(* Logix 5000 project; controller WWTP_SOLIDS_CLX vendor 1 type 14 code 54 rev 17.2; software revision 17.00; part 5 of 16 *)
(* tags used below, declared in another part *)
   Inp_RatePVBad : BOOL;   // 1=Rate PV Input Quality = Bad (fail)
   Inp_RatePVUncertain : BOOL;   // 1=Rate PV Input Quality = Uncertain
   Inp_QtyPVBad : BOOL;   // 1=Quantity PV Input Quality = Bad (fail)
   Inp_QtyPVUncertain : BOOL;   // 1=Quantity PV Input Quality = Uncertain
   Inp_CtrldEqpFault : BOOL;   // Controlled Equipment device or I/O status 0=OK, 1=fail
   Inp_Sim : BOOL;   // 1=Simulate working flowmeter; 0=use actual flowmeter
   Cfg_HasDribble : BOOL;   // 1=Slow to Dribble before complete, 0=use complete only
   Cfg_CalcRate : BOOL;   // 1=differentiate Inp_Qty to get rate, 0=use Inp_Rate
   Cfg_CalcQty : BOOL;   // 1=integrate Inp_Rate to get Quantity, 0=use Inp_Qty
   Cfg_PCmdClear : BOOL;   // 1=Clear Program Commands on receipt 0=Leave Set
   Cfg_HasOverTolAlm : BOOL;   // 1=Over Tolerance Alarm exists and will be checked
   Cfg_HasUnderTolAlm : BOOL;   // 1=Under Tolerance Alarm exists and will be checked
   Cfg_HasZeroFaultAlm : BOOL;   // 1=Zero Fault Alarm exists and will be checked
   Cfg_HasEqpFaultAlm : BOOL;   // 1=Equipment Fault Alarm exists and will be checked
   Cfg_OverTolResetReqd : BOOL;   // 1=Reset requied to clear Out of Tolerance High Alarm
   Cfg_UnderTolResetReqd : BOOL;   // 1=Reset required to clear Out of Tolerance Low Alarm
   Cfg_ZeroFaultResetReqd : BOOL;   // 1=Reset required to clear Zero Fault Alarm
   Cfg_EqpFaultResetReqd : BOOL;   // 1=Reset required to clear Equipment Fault Alarm
   Cfg_OverTolAckReqd : BOOL;   // 1=Acknowledge required for Out of Tolerance High Alarm
   Cfg_UnderTolAckReqd : BOOL;   // 1=Acknowledge required for Out of Tolerance Low Alarm
   Cfg_ZeroFaultAckReqd : BOOL;   // 1=Acknowledge required for Zero Fault Alarm
   Cfg_EqpFaultAckReqd : BOOL;   // 1=Acknowledge required for Equipment Fault Alarm
   Cfg_OverTolSeverity : SINT;   // Over Tolerance Alarm Severity 1=info, 2=warn, 3=excep, 4=fault
   Cfg_UnderTolSeverity : SINT;   // Under Tolerance Alarm Severity 1=info, 2=warn, 3=excep, 4=fault
   Cfg_ZeroFaultSeverity : SINT;   // Zero Fault Alarm Severity 1=info, 2=warn, 3=excep, 4=fault
   Cfg_EqpFaultSeverity : SINT;   // Equipment Fault Alarm Severity 1=info, 2=warn, 3=excep, 4=fault
   Cfg_MaxQty : REAL;   // Maximum allowed quantity to deliver (setpoint) (EU)
   Cfg_EUQtyMult : REAL;   // Rate to Quantity EU Multiplier (e.g., Gal to Bbl.)
   Cfg_Rollover : REAL;   // Quantity Rollover (e.g., total counts for pulse input)
   Cfg_CountsPerEU : REAL;   // Number of Counts in Inp_QtyPV which equal 1.0 EU
   Cfg_RateTime : REAL;   // Time factor for rate (60 for /min, 3600 for /hr) (Sec)
   Cfg_RateFiltTC : REAL;   // Filter Time Constant (sec) for calculated Rate
   Cfg_LoRateCutoff : REAL;   // Rate below which to report zero flow (Inp_RatePV untis)
   Cfg_SimRate : REAL;   // Rate at which to deliver when running in Simulation (EU/rate time)
   Cfg_SimDribbleRate : REAL;   // Rate at which to dribble when running in Simulation (EU/rate time)
   PCmd_OverTolAck : BOOL;   // Program Command to Acknowledge Out of Tolerance High Alarm
   PCmd_OverTolInhibit : BOOL;   // Program Command to Inhibit Out of Tolerance High Alarm
   PCmd_OverTolUninhibit : BOOL;   // Program Command to Uninhibit Out of Tolerance High Alarm
   PCmd_UnderTolAck : BOOL;   // Program Command to Acknowledge Out of Tolerance Low Alarm
   PCmd_UnderTolInhibit : BOOL;   // Program Command to Inhibit Out of Tolerance Low Alarm
   PCmd_UnderTolUninhibit : BOOL;   // Program Command to Uninhibit Out of Tolerance Low Alarm
   PCmd_ZeroFaultAck : BOOL;   // Program Command to Acknowledge Zero Fault Alarm
   PCmd_ZeroFaultInhibit : BOOL;   // Program Command to Inhibit Zero Fault Alarm
   PCmd_ZeroFaultUninhibit : BOOL;   // Program Command to Uninhibit Zero Fault Alarm
   PCmd_EqpFaultAck : BOOL;   // Program Command to Acknowledge Equipment Fault Alarm
   PCmd_EqpFaultInhibit : BOOL;   // Program Command to Inhibit Equipment Fault Alarm
   PCmd_EqpFaultUninhibit : BOOL;   // Program Command to Uninhibit Equipment Fault Alarm
   Out_RunFlow : BOOL;   // 1=Deliver at Full (fast) Flow
   Out_DribbleFlow : BOOL;   // 1=Deliver at Dribble (slow) Flow
   Out_StopFlow : BOOL;   // 1=Stop Delivery Equipment
   Out_RunTot : BOOL;   // 1=Run external totalizer (e.g. onboard flowmeter)
   Val_Qty : REAL;   // Quantity actually delivered (totalizer output) (EU)
   Val_SP : REAL;   // Amount to be delivered (Setpoint) (EU)
   Val_DribbleQty : REAL;   // Amount to be delivered at slow rate (EU)
   Val_Preact : REAL;   // Amount before SP at which flow will be stopped (EU)
   Val_Notify : SINT;   // Current Alarm Level and Acknowledgement (enumeration)
   Sts_Cleared : BOOL;   // 1=Totalizer Clear completed
   Sts_TotRunning : BOOL;   // 1=Totalizer Running, 0=Totalizer Stopped
   Sts_FlowRunning : BOOL;   // 1=Flow is Running (Out_Run is ON)
   Sts_FlowDribble : BOOL;   // 1=Flow is slowed to Dribble (Out_Dribble is ON)
   Sts_FlowStopped : BOOL;   // 1=Flow is Stopped (Out_Stop is ON)
   Sts_Bumping : BOOL;   // 1=Bump flow (timed) is active
   Sts_Complete : BOOL;   // 1=Total Delivered > (SP - Preact)
   Sts_Available : BOOL;   // 1=Dosing available for control by automation (Prog)
   Sts_QtyBad : BOOL;   // 1=Quantity Value is Bad (PV Fail)
   Sts_QtyUncertain : BOOL;   // 1=Quantity Value is Uncertain
   Sts_RateBad : BOOL;   // 1=Rate Value is Bad (PV Fail)
   Sts_RateUncertain : BOOL;   // 1=Rate Value is Uncertain
   Sts_Err : BOOL;   // 1=Error: Bad Configuration, see detail Err bits for reason
   Err_EU : BOOL;   // 1=Error: Cfg_CountsPerEU, Cfg_EUQtyMult or Cfg_Rollowver invalid
   Err_Rate : BOOL;   // 1=Error: Cfg_RateFiltTC or Cfg_RateTime invalid
   Err_Cutoff : BOOL;   // 1=Error: Cfg_LoRateCutoff invalid
   Err_Limit : BOOL;   // 1=Error: Cfg_MaxQty invalid
   Err_Sim : BOOL;   // 1=Error: Cfg_SimDribbleRate or Cfg_SimRate invalid
   Err_Timer : BOOL;   // 1=Error: Cfg_BumpT or Cfg_ClearPulseT (use 0.0 to 2147483.647)
   Err_Alarm : BOOL;   // 1=Error: Alarm Severity Cfg Invalid
   Sts_Maint : BOOL;   // 1=Mode is Maintenance (supersedes Prog, Oper)
   Sts_Prog : BOOL;   // 1=Mode is Program (auto)
   Sts_Oper : BOOL;   // 1=Mode is Operator (manual)
   Sts_ProgOperLock : BOOL;   // 1=Program or Operator has requested Mode Lock
   Sts_OverTol : BOOL;   // 1=Delivery Out of Tolerance High
   Alm_OverTol : BOOL;   // 1=Delivery Out of Tolerance High Alarm
   Ack_OverTol : BOOL;   // 1=Out of Tolerance High Alarm has been acknowledged
   Sts_OverTolDisabled : BOOL;   // 1=Out of Tolerance High Alarm has been disabled (will not be sent)
   Sts_OverTolInhibited : BOOL;   // 1=Out of Tolerance High Alarm has been inhibited by logic
   Sts_OverTolSuppressed : BOOL;   // 1=Out of Tolerance High Alarm has been suppressed (logged only)
   Sts_UnderTol : BOOL;   // 1=Delivery Out of Tolerance Low
   Alm_UnderTol : BOOL;   // 1=Delivery Out of Tolerance Low Alarm
   Ack_UnderTol : BOOL;   // 1=Out of Tolerance Low Alarm has been acknowledged
   Sts_UnderTolDisabled : BOOL;   // 1=Out of Tolerance Low Alarm has been disabled (will not be sent)
   Sts_UnderTolInhibited : BOOL;   // 1=Out of Tolerance Low Alarm has been inhibited by logic
   Sts_UnderTolSuppressed : BOOL;   // 1=Out of Tolerance Low Alarm has been suppressed (logged only)
   Sts_ZeroFault : BOOL;   // 1=Total did not clear or unexpected flow
   Alm_ZeroFault : BOOL;   // 1=Warning: Total did not clear or still flowing
   Ack_ZeroFault : BOOL;   // 1=Zero Fault Alarm has been acknowledged
   Sts_ZeroFaultDisabled : BOOL;   // 1=Zero Fault Alarm is Disabled (not saved or sent)
   Sts_ZeroFaultInhibited : BOOL;   // 1=Zero Fault Alarm has been inhibited by logic
   Sts_ZeroFaultSuppressed : BOOL;   // 1=Zero Fault Alarm has been suppressed (logged only)
   Sts_EqpFault : BOOL;   // 1=Equipment Fault Detected
   Alm_EqpFault : BOOL;   // 1=Equipment Fault Alarm
   Ack_EqpFault : BOOL;   // 1=Equipment Fault Alarm has been acknowledged
   Sts_EqpFaultDisabled : BOOL;   // 1=Equipment Fault Alarm is Disabled (not saved or sent)
   Sts_EqpFaultInhibited : BOOL;   // 1=Equipment Fault Alarm has been inhibited by logic
   Sts_EqpFaultSuppressed : BOOL;   // 1=Equipment Fault Alarm has been suppressed (logged only)
   Rdy_ClearTot : BOOL;   // 1=Ready for OCmd_ClearTot (enables button)
   Rdy_StartTot : BOOL;   // 1=Ready for OCmd_StartTot (enables button)
   Rdy_StopTot : BOOL;   // 1=Ready for OCmd_StopTot (enables button)
   Rdy_StartFlow : BOOL;   // 1=Ready for OCmd_StartFlow (enables button)
   Rdy_StopFlow : BOOL;   // 1=Ready for OCmd_StopFlow (enables button)
   Rdy_CheckTol : BOOL;   // 1-Ready for OCmd_CheckTol (enables button)
   Rdy_Bump : BOOL;   // 1=Ready for OCmd_Bump (enables button)
   Rdy_Reset : BOOL;   // 1=Ready for OCmd_Reset (enables button)
   Wrk_Notify : DINT;   // Buffer for building Val_Notify
   Mode : P_Mode;   // Analog Input Mode Selection
   Wrk_ClearTot : BOOL;   // Request to Clear Total received
   ZeroFault : P_Alarm;   // Rate Not Zero when Expected Alarm
   UnderTol : P_Alarm;   // Final Quantity Below Low Tolerance Alarm
   OverTol : P_Alarm;   // Final Quantity Above High Tolerance Alarm
   EqpFault : P_Alarm;   // Equipment (Sensor, Controlled Equip.) Fault Alarm
   Wrk_RunFlow : BOOL;   // 1=Flow (full)( should be running
   Wrk_RunTot : BOOL;   // 1=Totalizaer should be ruuuning
   Wrk_BumpFlow : BOOL;   // Operator requested bump flow to make up Under Tolerance
   Wrk_BumpT : TIMER;   // Bump Timer for shot of flow to make up Under Tolerance
   Wrk_ClearPulseT : TIMER;   // Time to pulse Out_Clear to clear external timer
   Wrk_LoOrderTot : REAL;   // Fractional Amount of Totalizer (low-order of cascaded registers)
   Wrk_HiOrderTot : DINT;   // Integer Amount of Totalizer (high-order of cascaded registers)
   Wrk_RateInfNaN : BOOL;   // Rate PV is Infinite or NaN
   Wrk_QtyInfNaN : BOOL;   // Quantity PV is Infinite or NaN
(* P_DoseFM, continued *)

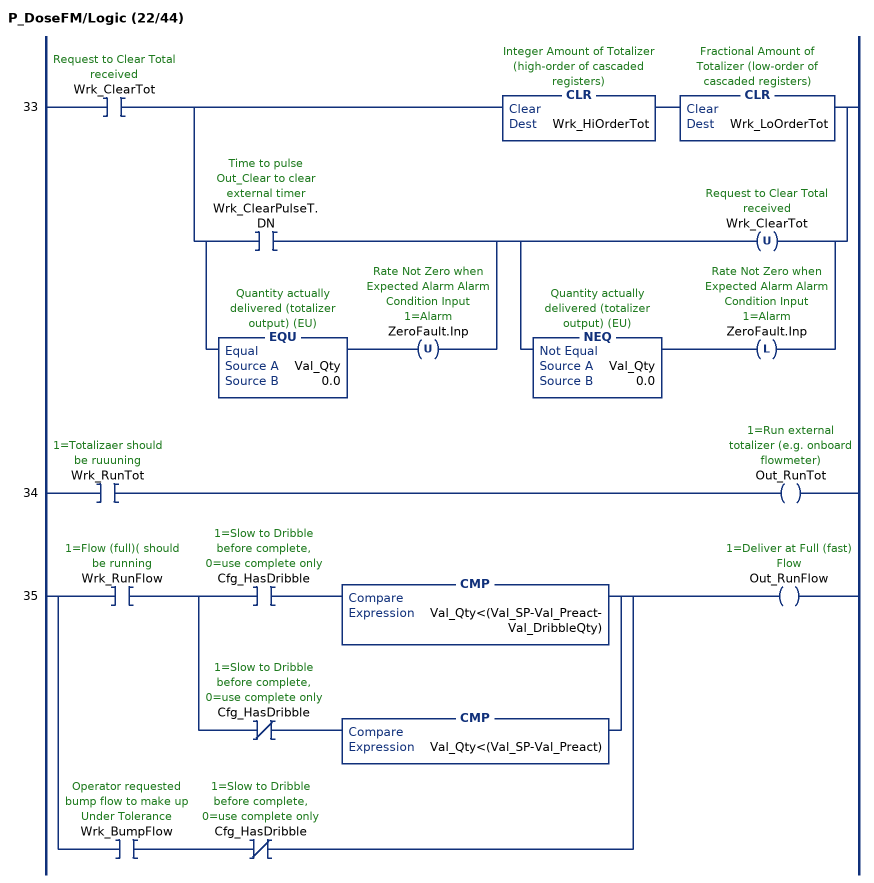
   [picture p88: P_DoseFM/Logic rungs 33-35]
   33: XIC(Wrk_ClearTot)[CLR(Wrk_HiOrderTot) CLR(Wrk_LoOrderTot) ,[XIC(Wrk_ClearPulseT.DN) ,EQU(Val_Qty,0.0) OTU(ZeroFault.Inp) ] [OTU(Wrk_ClearTot) ,NEQ(Val_Qty,0.0) OTL(ZeroFault.Inp) ] ];
   34: XIC(Wrk_RunTot)OTE(Out_RunTot);
   35: [XIC(Wrk_RunFlow) [XIC(Cfg_HasDribble) CMP(Val_Qty<(Val_SP-Val_Preact-Val_DribbleQty)) ,XIO(Cfg_HasDribble) CMP(Val_Qty<(Val_SP-Val_Preact)) ] ,XIC(Wrk_BumpFlow) XIO(Cfg_HasDribble) ]OTE(Out_RunFlow);
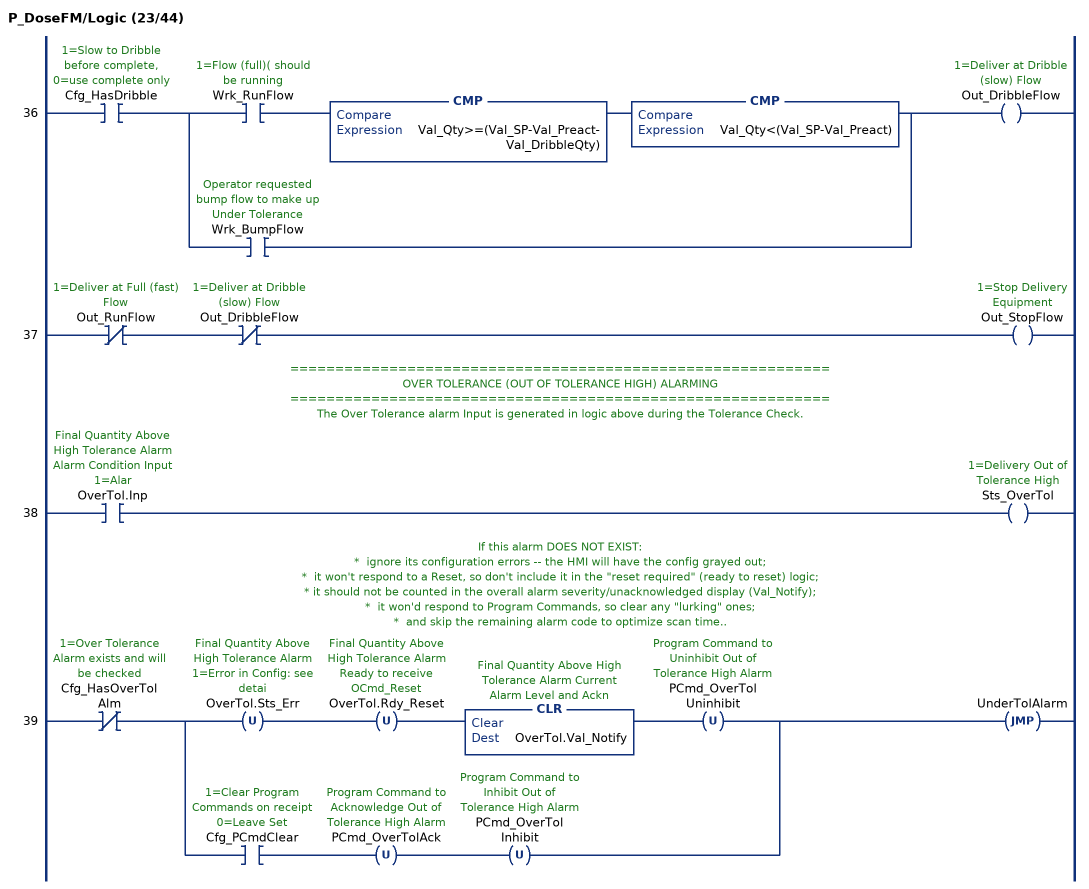
   36: XIC(Cfg_HasDribble)[XIC(Wrk_RunFlow) CMP(Val_Qty>=(Val_SP-Val_Preact-Val_DribbleQty)) CMP(Val_Qty<(Val_SP-Val_Preact)) ,XIC(Wrk_BumpFlow) ]OTE(Out_DribbleFlow);
   37: XIO(Out_RunFlow)XIO(Out_DribbleFlow)OTE(Out_StopFlow);
   // ============================================================
   // OVER TOLERANCE (OUT OF TOLERANCE HIGH) ALARMING
   // ============================================================
   // The Over Tolerance alarm Input is generated in logic above during the Tolerance Check.
   38: XIC(OverTol.Inp)OTE(Sts_OverTol);
   // If this alarm DOES NOT EXIST:
   // *  ignore its configuration errors -- the HMI will have the config grayed out;
   // *  it won't respond to a Reset, so don't include it in the "reset required" (ready to reset) logic;
   // * it should not be counted in the overall alarm severity/unacknowledged display (Val_Notify);
   // *  it won'd respond to Program Commands, so clear any "lurking" ones;
   // *  and skip the remaining alarm code to optimize scan time..
   39: XIO(Cfg_HasOverTolAlm)[OTU(OverTol.Sts_Err) OTU(OverTol.Rdy_Reset) CLR(OverTol.Val_Notify) OTU(PCmd_OverTolUninhibit) ,XIC(Cfg_PCmdClear) OTU(PCmd_OverTolAck) OTU(PCmd_OverTolInhibit) ]JMP(UnderTolAlarm);
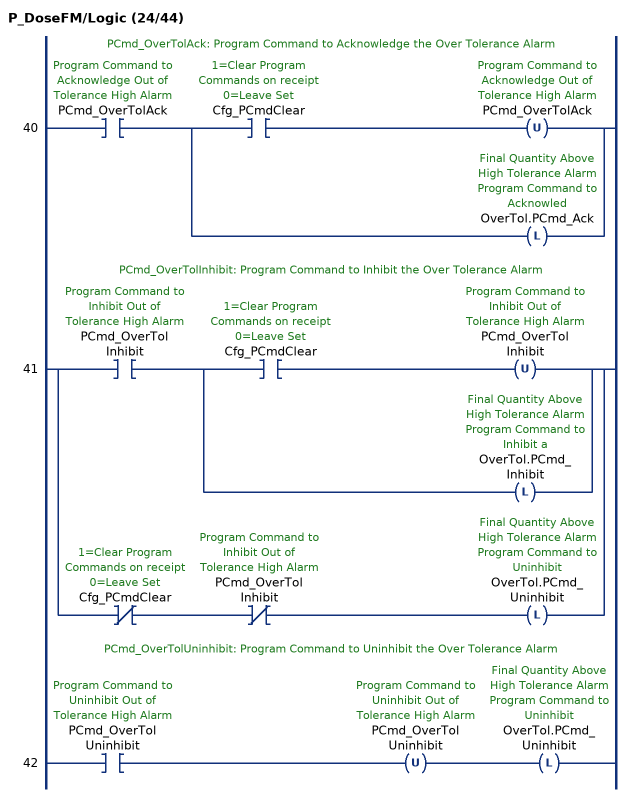
   // PCmd_OverTolAck: Program Command to Acknowledge the Over Tolerance Alarm
   40: XIC(PCmd_OverTolAck)[XIC(Cfg_PCmdClear) OTU(PCmd_OverTolAck) ,OTL(OverTol.PCmd_Ack) ];
   // PCmd_OverTolInhibit: Program Command to Inhibit the Over Tolerance Alarm
   41: [XIC(PCmd_OverTolInhibit) [XIC(Cfg_PCmdClear) OTU(PCmd_OverTolInhibit) ,OTL(OverTol.PCmd_Inhibit) ] ,XIO(Cfg_PCmdClear) XIO(PCmd_OverTolInhibit) OTL(OverTol.PCmd_Uninhibit) ];
   // PCmd_OverTolUninhibit: Program Command to Uninhibit the Over Tolerance Alarm
   42: XIC(PCmd_OverTolUninhibit)OTU(PCmd_OverTolUninhibit)OTL(OverTol.PCmd_Uninhibit);
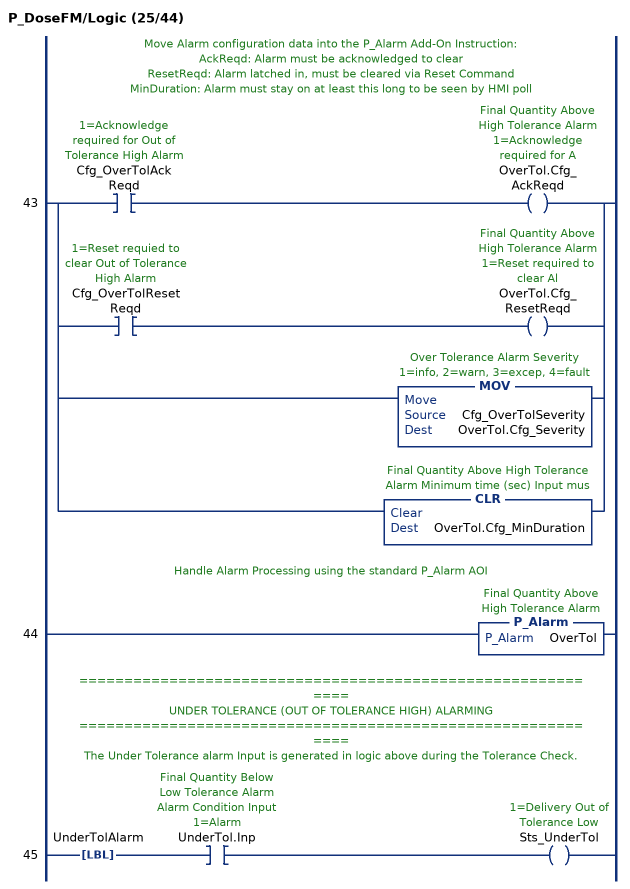
   // Move Alarm configuration data into the P_Alarm Add-On Instruction:
   // AckReqd: Alarm must be acknowledged to clear
   // ResetReqd: Alarm latched in, must be cleared via Reset Command
   // MinDuration: Alarm must stay on at least this long to be seen by HMI poll
   43: [XIC(Cfg_OverTolAckReqd) OTE(OverTol.Cfg_AckReqd) ,XIC(Cfg_OverTolResetReqd) OTE(OverTol.Cfg_ResetReqd) ,MOV(Cfg_OverTolSeverity,OverTol.Cfg_Severity) ,CLR(OverTol.Cfg_MinDuration) ];
   // Handle Alarm Processing using the standard P_Alarm AOI
   44: P_Alarm(OverTol);
   // ============================================================
   // UNDER TOLERANCE (OUT OF TOLERANCE HIGH) ALARMING
   // ============================================================
   // The Under Tolerance alarm Input is generated in logic above during the Tolerance Check.
   45: LBL(UnderTolAlarm)XIC(UnderTol.Inp)OTE(Sts_UnderTol);
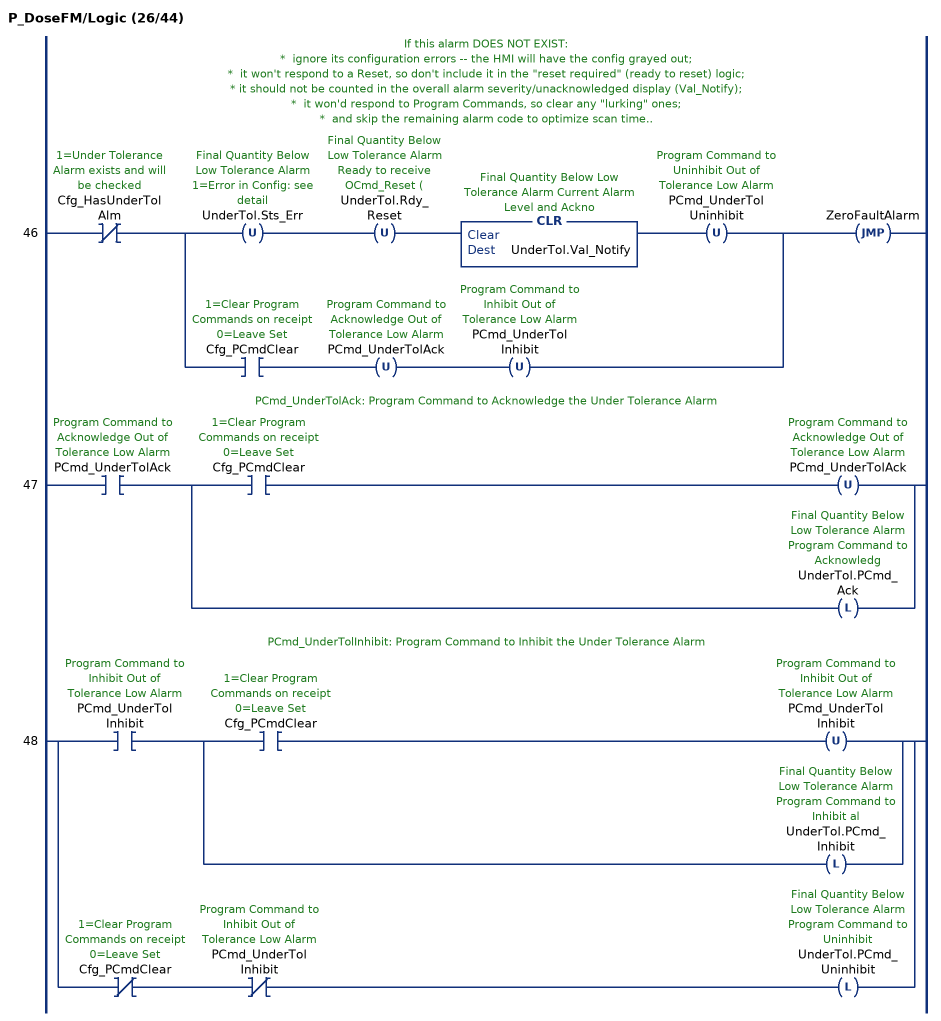
   // If this alarm DOES NOT EXIST:
   // *  ignore its configuration errors -- the HMI will have the config grayed out;
   // *  it won't respond to a Reset, so don't include it in the "reset required" (ready to reset) logic;
   // * it should not be counted in the overall alarm severity/unacknowledged display (Val_Notify);
   // *  it won'd respond to Program Commands, so clear any "lurking" ones;
   // *  and skip the remaining alarm code to optimize scan time..
   46: XIO(Cfg_HasUnderTolAlm)[OTU(UnderTol.Sts_Err) OTU(UnderTol.Rdy_Reset) CLR(UnderTol.Val_Notify) OTU(PCmd_UnderTolUninhibit) ,XIC(Cfg_PCmdClear) OTU(PCmd_UnderTolAck) OTU(PCmd_UnderTolInhibit) ]JMP(ZeroFaultAlarm);
   // PCmd_UnderTolAck: Program Command to Acknowledge the Under Tolerance Alarm
   47: XIC(PCmd_UnderTolAck)[XIC(Cfg_PCmdClear) OTU(PCmd_UnderTolAck) ,OTL(UnderTol.PCmd_Ack) ];
   // PCmd_UnderTolInhibit: Program Command to Inhibit the Under Tolerance Alarm
   48: [XIC(PCmd_UnderTolInhibit) [XIC(Cfg_PCmdClear) OTU(PCmd_UnderTolInhibit) ,OTL(UnderTol.PCmd_Inhibit) ] ,XIO(Cfg_PCmdClear) XIO(PCmd_UnderTolInhibit) OTL(UnderTol.PCmd_Uninhibit) ];
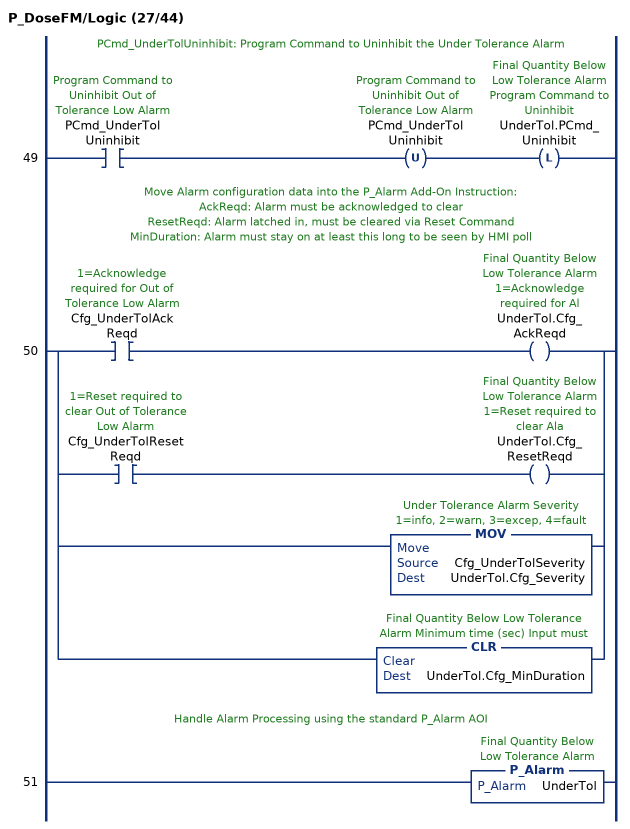
   // PCmd_UnderTolUninhibit: Program Command to Uninhibit the Under Tolerance Alarm
   49: XIC(PCmd_UnderTolUninhibit)OTU(PCmd_UnderTolUninhibit)OTL(UnderTol.PCmd_Uninhibit);
   // Move Alarm configuration data into the P_Alarm Add-On Instruction:
   // AckReqd: Alarm must be acknowledged to clear
   // ResetReqd: Alarm latched in, must be cleared via Reset Command
   // MinDuration: Alarm must stay on at least this long to be seen by HMI poll
   50: [XIC(Cfg_UnderTolAckReqd) OTE(UnderTol.Cfg_AckReqd) ,XIC(Cfg_UnderTolResetReqd) OTE(UnderTol.Cfg_ResetReqd) ,MOV(Cfg_UnderTolSeverity,UnderTol.Cfg_Severity) ,CLR(UnderTol.Cfg_MinDuration) ];
   // Handle Alarm Processing using the standard P_Alarm AOI
   51: P_Alarm(UnderTol);
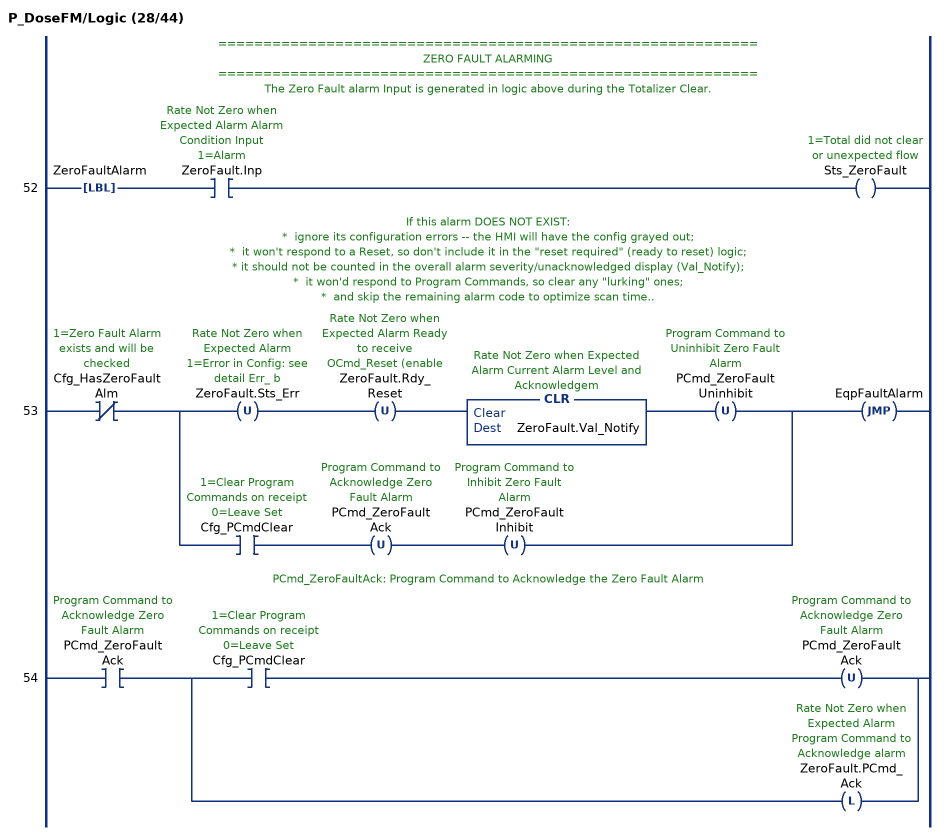
   // ============================================================
   // ZERO FAULT ALARMING
   // ============================================================
   // The Zero Fault alarm Input is generated in logic above during the Totalizer Clear.
   52: LBL(ZeroFaultAlarm)XIC(ZeroFault.Inp)OTE(Sts_ZeroFault);
   // If this alarm DOES NOT EXIST:
   // *  ignore its configuration errors -- the HMI will have the config grayed out;
   // *  it won't respond to a Reset, so don't include it in the "reset required" (ready to reset) logic;
   // * it should not be counted in the overall alarm severity/unacknowledged display (Val_Notify);
   // *  it won'd respond to Program Commands, so clear any "lurking" ones;
   // *  and skip the remaining alarm code to optimize scan time..
   53: XIO(Cfg_HasZeroFaultAlm)[OTU(ZeroFault.Sts_Err) OTU(ZeroFault.Rdy_Reset) CLR(ZeroFault.Val_Notify) OTU(PCmd_ZeroFaultUninhibit) ,XIC(Cfg_PCmdClear) OTU(PCmd_ZeroFaultAck) OTU(PCmd_ZeroFaultInhibit) ]JMP(EqpFaultAlarm);
   // PCmd_ZeroFaultAck: Program Command to Acknowledge the Zero Fault Alarm
   54: XIC(PCmd_ZeroFaultAck)[XIC(Cfg_PCmdClear) OTU(PCmd_ZeroFaultAck) ,OTL(ZeroFault.PCmd_Ack) ];
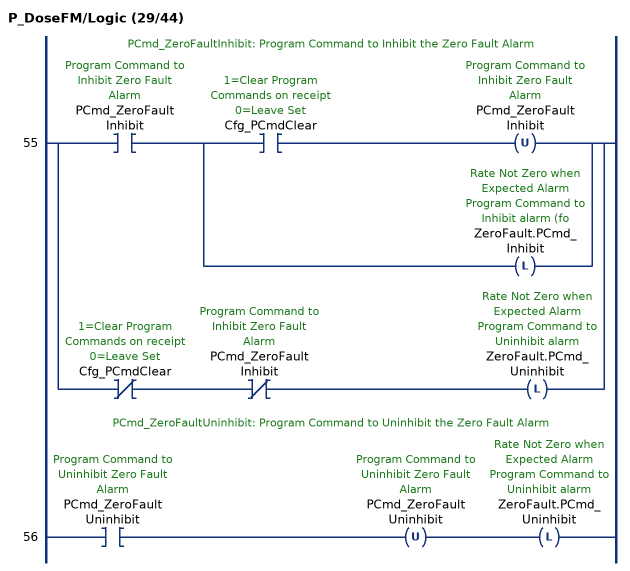
   // PCmd_ZeroFaultInhibit: Program Command to Inhibit the Zero Fault Alarm
   55: [XIC(PCmd_ZeroFaultInhibit) [XIC(Cfg_PCmdClear) OTU(PCmd_ZeroFaultInhibit) ,OTL(ZeroFault.PCmd_Inhibit) ] ,XIO(Cfg_PCmdClear) XIO(PCmd_ZeroFaultInhibit) OTL(ZeroFault.PCmd_Uninhibit) ];
   // PCmd_ZeroFaultUninhibit: Program Command to Uninhibit the Zero Fault Alarm
   56: XIC(PCmd_ZeroFaultUninhibit)OTU(PCmd_ZeroFaultUninhibit)OTL(ZeroFault.PCmd_Uninhibit);
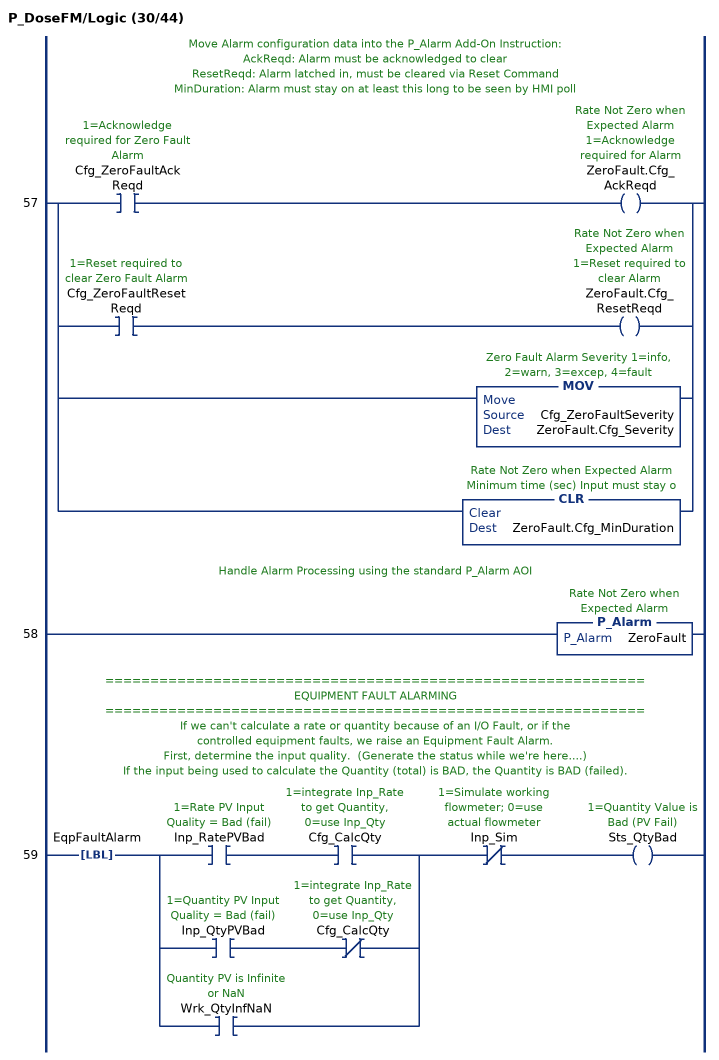
   // Move Alarm configuration data into the P_Alarm Add-On Instruction:
   // AckReqd: Alarm must be acknowledged to clear
   // ResetReqd: Alarm latched in, must be cleared via Reset Command
   // MinDuration: Alarm must stay on at least this long to be seen by HMI poll
   57: [XIC(Cfg_ZeroFaultAckReqd) OTE(ZeroFault.Cfg_AckReqd) ,XIC(Cfg_ZeroFaultResetReqd) OTE(ZeroFault.Cfg_ResetReqd) ,MOV(Cfg_ZeroFaultSeverity,ZeroFault.Cfg_Severity) ,CLR(ZeroFault.Cfg_MinDuration) ];
   // Handle Alarm Processing using the standard P_Alarm AOI
   58: P_Alarm(ZeroFault);
   // ============================================================
   // EQUIPMENT FAULT ALARMING
   // ============================================================
   // If we can't calculate a rate or quantity because of an I/O Fault, or if the
   // controlled equipment faults, we raise an Equipment Fault Alarm.
   // First, determine the input quality.  (Generate the status while we're here....)
   // If the input being used to calculate the Quantity (total) is BAD, the Quantity is BAD (failed).
   59: LBL(EqpFaultAlarm)[XIC(Inp_RatePVBad) XIC(Cfg_CalcQty) ,XIC(Inp_QtyPVBad) XIO(Cfg_CalcQty) ,XIC(Wrk_QtyInfNaN) ]XIO(Inp_Sim)OTE(Sts_QtyBad);
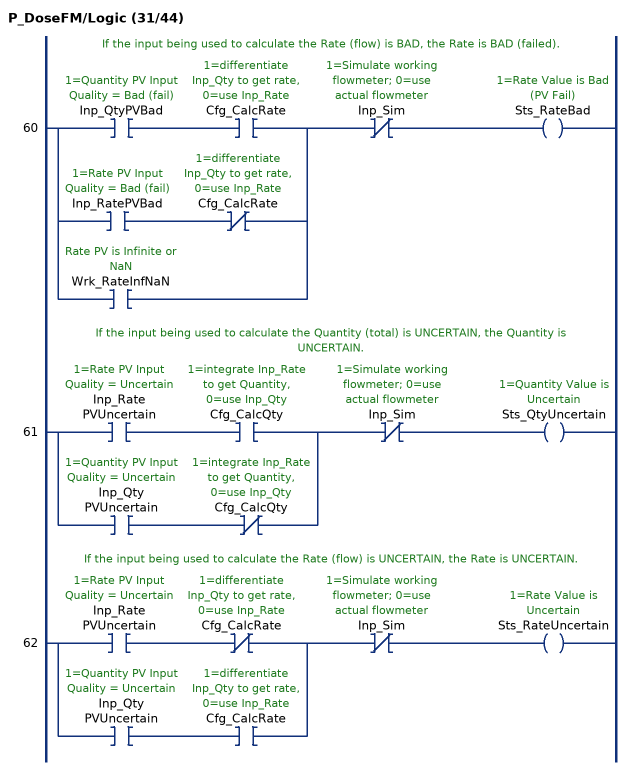
   // If the input being used to calculate the Rate (flow) is BAD, the Rate is BAD (failed).
   60: [XIC(Inp_QtyPVBad) XIC(Cfg_CalcRate) ,XIC(Inp_RatePVBad) XIO(Cfg_CalcRate) ,XIC(Wrk_RateInfNaN) ]XIO(Inp_Sim)OTE(Sts_RateBad);
   // If the input being used to calculate the Quantity (total) is UNCERTAIN, the Quantity is UNCERTAIN.
   61: [XIC(Inp_RatePVUncertain) XIC(Cfg_CalcQty) ,XIC(Inp_QtyPVUncertain) XIO(Cfg_CalcQty) ]XIO(Inp_Sim)OTE(Sts_QtyUncertain);
   // If the input being used to calculate the Rate (flow) is UNCERTAIN, the Rate is UNCERTAIN.
   62: [XIC(Inp_RatePVUncertain) XIO(Cfg_CalcRate) ,XIC(Inp_QtyPVUncertain) XIC(Cfg_CalcRate) ]XIO(Inp_Sim)OTE(Sts_RateUncertain);
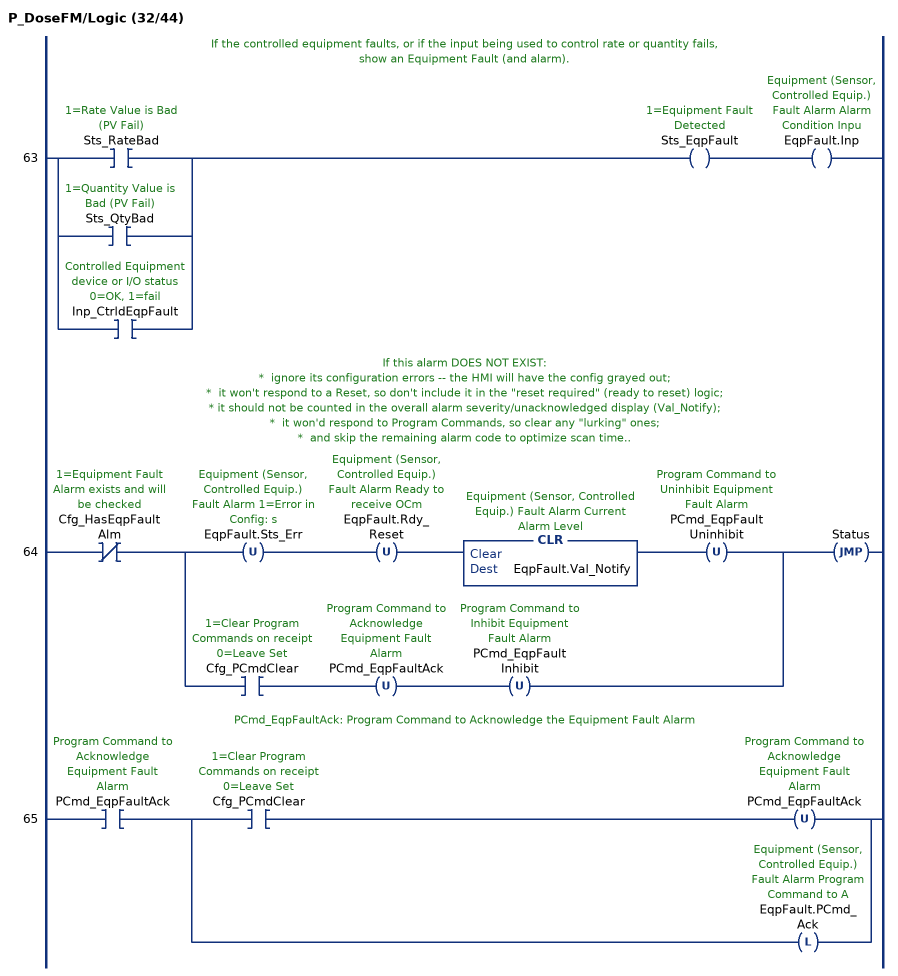
   // If the controlled equipment faults, or if the input being used to control rate or quantity fails,
   // show an Equipment Fault (and alarm).
   63: [XIC(Sts_RateBad) ,XIC(Sts_QtyBad) ,XIC(Inp_CtrldEqpFault) ]OTE(Sts_EqpFault)OTE(EqpFault.Inp);
   // If this alarm DOES NOT EXIST:
   // *  ignore its configuration errors -- the HMI will have the config grayed out;
   // *  it won't respond to a Reset, so don't include it in the "reset required" (ready to reset) logic;
   // * it should not be counted in the overall alarm severity/unacknowledged display (Val_Notify);
   // *  it won'd respond to Program Commands, so clear any "lurking" ones;
   // *  and skip the remaining alarm code to optimize scan time..
   64: XIO(Cfg_HasEqpFaultAlm)[OTU(EqpFault.Sts_Err) OTU(EqpFault.Rdy_Reset) CLR(EqpFault.Val_Notify) OTU(PCmd_EqpFaultUninhibit) ,XIC(Cfg_PCmdClear) OTU(PCmd_EqpFaultAck) OTU(PCmd_EqpFaultInhibit) ]JMP(Status);
   // PCmd_EqpFaultAck: Program Command to Acknowledge the Equipment Fault Alarm
   65: XIC(PCmd_EqpFaultAck)[XIC(Cfg_PCmdClear) OTU(PCmd_EqpFaultAck) ,OTL(EqpFault.PCmd_Ack) ];
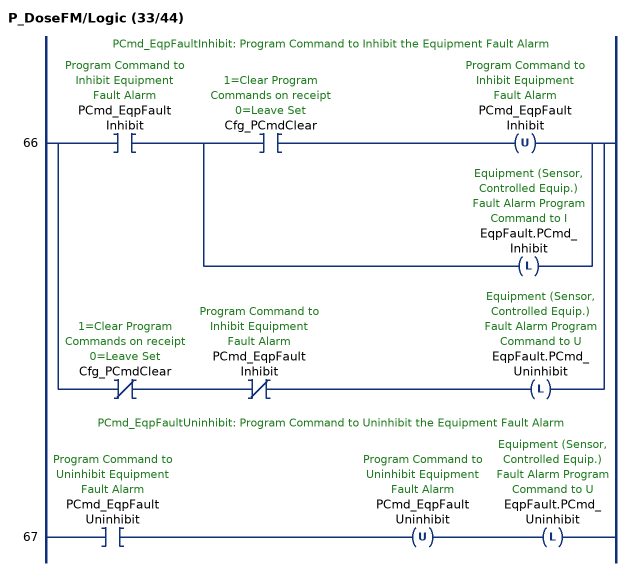
   // PCmd_EqpFaultInhibit: Program Command to Inhibit the Equipment Fault Alarm
   66: [XIC(PCmd_EqpFaultInhibit) [XIC(Cfg_PCmdClear) OTU(PCmd_EqpFaultInhibit) ,OTL(EqpFault.PCmd_Inhibit) ] ,XIO(Cfg_PCmdClear) XIO(PCmd_EqpFaultInhibit) OTL(EqpFault.PCmd_Uninhibit) ];
   // PCmd_EqpFaultUninhibit: Program Command to Uninhibit the Equipment Fault Alarm
   67: XIC(PCmd_EqpFaultUninhibit)OTU(PCmd_EqpFaultUninhibit)OTL(EqpFault.PCmd_Uninhibit);
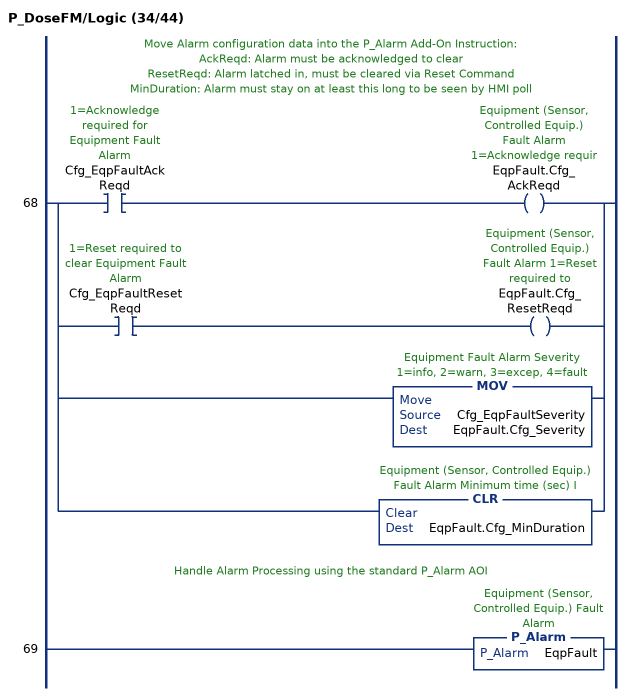
   // Move Alarm configuration data into the P_Alarm Add-On Instruction:
   // AckReqd: Alarm must be acknowledged to clear
   // ResetReqd: Alarm latched in, must be cleared via Reset Command
   // MinDuration: Alarm must stay on at least this long to be seen by HMI poll
   68: [XIC(Cfg_EqpFaultAckReqd) OTE(EqpFault.Cfg_AckReqd) ,XIC(Cfg_EqpFaultResetReqd) OTE(EqpFault.Cfg_ResetReqd) ,MOV(Cfg_EqpFaultSeverity,EqpFault.Cfg_Severity) ,CLR(EqpFault.Cfg_MinDuration) ];
   // Handle Alarm Processing using the standard P_Alarm AOI
   69: P_Alarm(EqpFault);
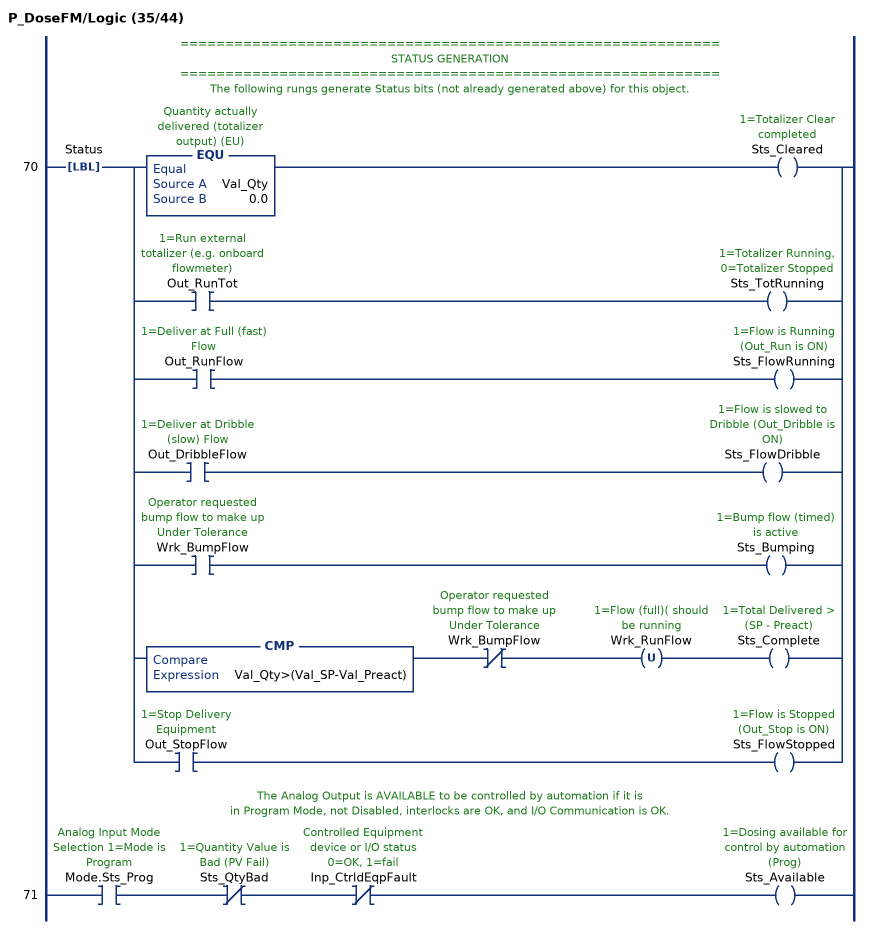
   // ============================================================
   // STATUS GENERATION
   // ============================================================
   // The following rungs generate Status bits (not already generated above) for this object.
   70: LBL(Status)[EQU(Val_Qty,0.0) OTE(Sts_Cleared) ,XIC(Out_RunTot) OTE(Sts_TotRunning) ,XIC(Out_RunFlow) OTE(Sts_FlowRunning) ,XIC(Out_DribbleFlow) OTE(Sts_FlowDribble) ,XIC(Wrk_BumpFlow) OTE(Sts_Bumping) ,CMP(Val_Qty>(Val_SP-Val_Preact)) XIO(Wrk_BumpFlow) OTU(Wrk_RunFlow) OTE(Sts_Complete) ,XIC(Out_StopFlow) OTE(Sts_FlowStopped) ];
   // The Analog Output is AVAILABLE to be controlled by automation if it is
   // in Program Mode, not Disabled, interlocks are OK, and I/O Communication is OK.
   71: XIC(Mode.Sts_Prog)XIO(Sts_QtyBad)XIO(Inp_CtrldEqpFault)OTE(Sts_Available);
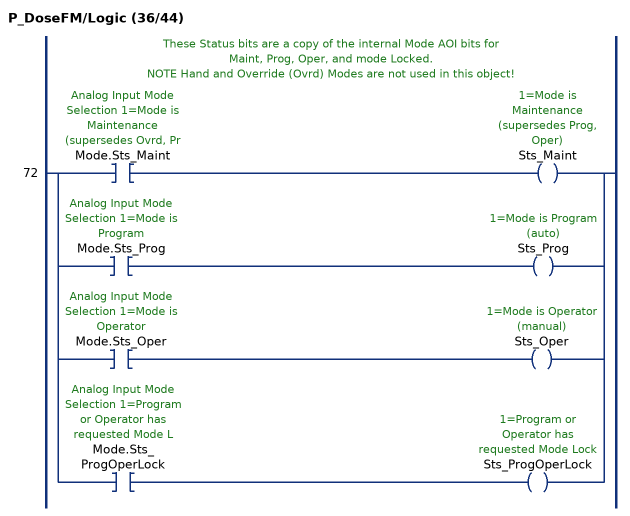
   // These Status bits are a copy of the internal Mode AOI bits for
   // Maint, Prog, Oper, and mode Locked.
   // NOTE Hand and Override (Ovrd) Modes are not used in this object!
   72: [XIC(Mode.Sts_Maint) OTE(Sts_Maint) ,XIC(Mode.Sts_Prog) OTE(Sts_Prog) ,XIC(Mode.Sts_Oper) OTE(Sts_Oper) ,XIC(Mode.Sts_ProgOperLock) OTE(Sts_ProgOperLock) ];
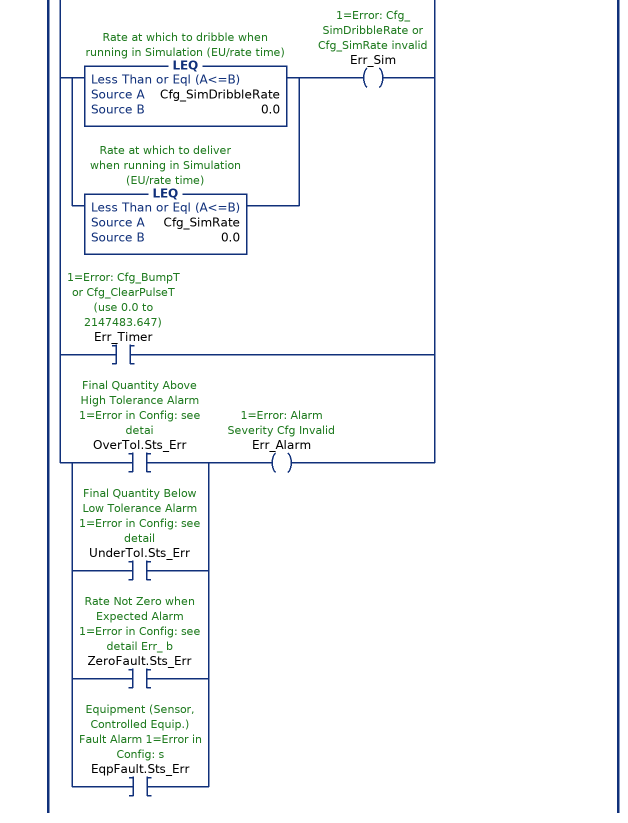
   // This rung handles the reports of all Error (Bad Configuration) Status.
   // Individual bits are provided for various status:
   // Invalid Engineering Units Scaling configs
   // Invalid Rate calculation configs
   // Invalid Limit configs
   // Invalid Simulation configs
   // Invalid Timer configs (determined in Configuration section above)
   // Then a summary Error Status is provided, simply an OR of the individual bits.
   73: [[LEQ(Cfg_CountsPerEU,0.0) ,LEQ(Cfg_EUQtyMult,0.0) ,LES(Cfg_Rollover,0.0) ] OTE(Err_EU) ,[LES(Cfg_RateFiltTC,0.0) ,LEQ(Cfg_RateTime,0.0) ] OTE(Err_Rate) ,LES(Cfg_LoRateCutoff,0.0) OTE(Err_Cutoff) ,LEQ(Cfg_MaxQty,0.0) OTE(Err_Limit) ,[LEQ(Cfg_SimDribbleRate,0.0) ,LEQ(Cfg_SimRate,0.0) ] OTE(Err_Sim) ,XIC(Err_Timer) ,[XIC(OverTol.Sts_Err) ,XIC(UnderTol.Sts_Err) ,XIC(ZeroFault.Sts_Err) ,XIC(EqpFault.Sts_Err) ] OTE(Err_Alarm) ]OTE(Sts_Err);
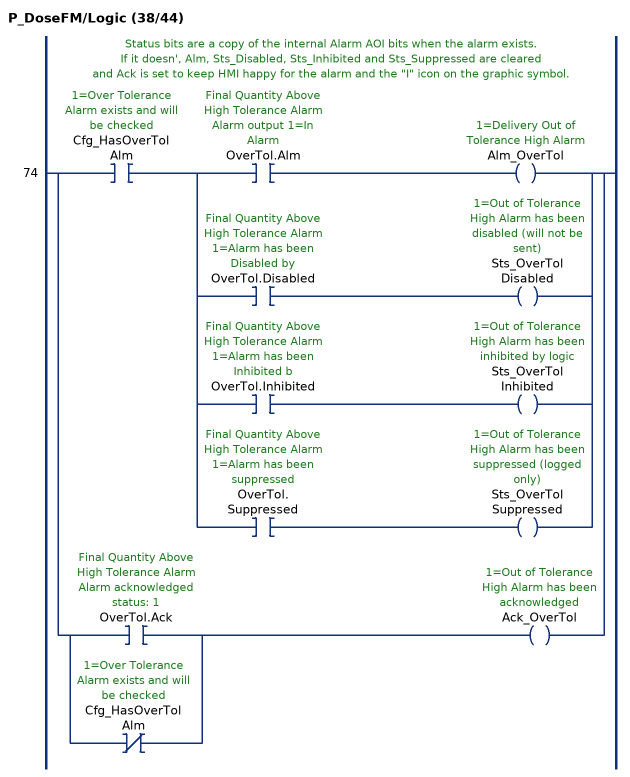
   // Status bits are a copy of the internal Alarm AOI bits when the alarm exists.
   // If it doesn', Alm, Sts_Disabled, Sts_Inhibited and Sts_Suppressed are cleared
   // and Ack is set to keep HMI happy for the alarm and the "I" icon on the graphic symbol.
   74: [XIC(Cfg_HasOverTolAlm) [XIC(OverTol.Alm) OTE(Alm_OverTol) ,XIC(OverTol.Disabled) OTE(Sts_OverTolDisabled) ,XIC(OverTol.Inhibited) OTE(Sts_OverTolInhibited) ,XIC(OverTol.Suppressed) OTE(Sts_OverTolSuppressed) ] ,[XIC(OverTol.Ack) ,XIO(Cfg_HasOverTolAlm) ] OTE(Ack_OverTol) ];
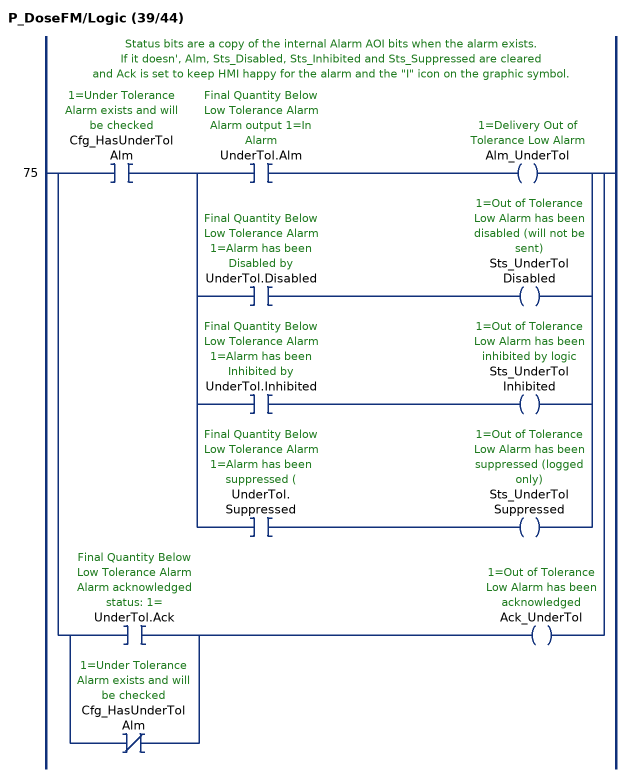
   // Status bits are a copy of the internal Alarm AOI bits when the alarm exists.
   // If it doesn', Alm, Sts_Disabled, Sts_Inhibited and Sts_Suppressed are cleared
   // and Ack is set to keep HMI happy for the alarm and the "I" icon on the graphic symbol.
   75: [XIC(Cfg_HasUnderTolAlm) [XIC(UnderTol.Alm) OTE(Alm_UnderTol) ,XIC(UnderTol.Disabled) OTE(Sts_UnderTolDisabled) ,XIC(UnderTol.Inhibited) OTE(Sts_UnderTolInhibited) ,XIC(UnderTol.Suppressed) OTE(Sts_UnderTolSuppressed) ] ,[XIC(UnderTol.Ack) ,XIO(Cfg_HasUnderTolAlm) ] OTE(Ack_UnderTol) ];
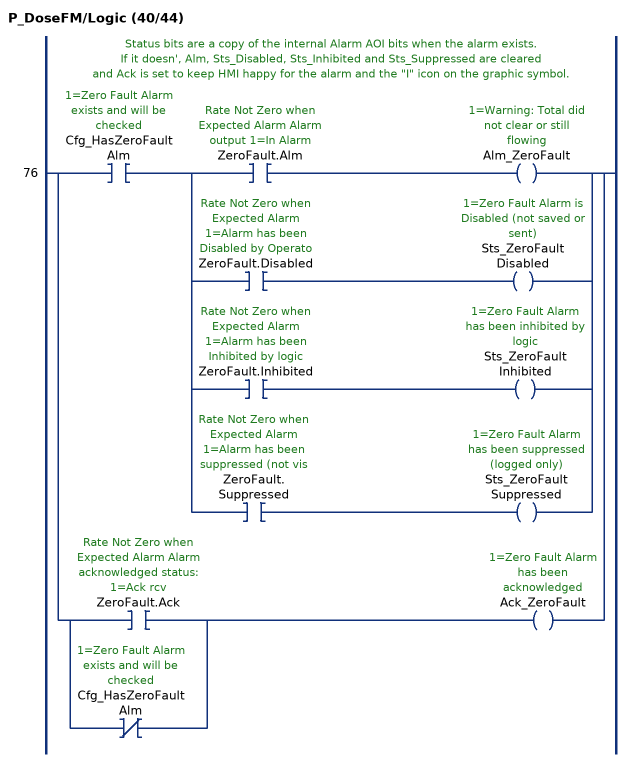
   // Status bits are a copy of the internal Alarm AOI bits when the alarm exists.
   // If it doesn', Alm, Sts_Disabled, Sts_Inhibited and Sts_Suppressed are cleared
   // and Ack is set to keep HMI happy for the alarm and the "I" icon on the graphic symbol.
   76: [XIC(Cfg_HasZeroFaultAlm) [XIC(ZeroFault.Alm) OTE(Alm_ZeroFault) ,XIC(ZeroFault.Disabled) OTE(Sts_ZeroFaultDisabled) ,XIC(ZeroFault.Inhibited) OTE(Sts_ZeroFaultInhibited) ,XIC(ZeroFault.Suppressed) OTE(Sts_ZeroFaultSuppressed) ] ,[XIC(ZeroFault.Ack) ,XIO(Cfg_HasZeroFaultAlm) ] OTE(Ack_ZeroFault) ];
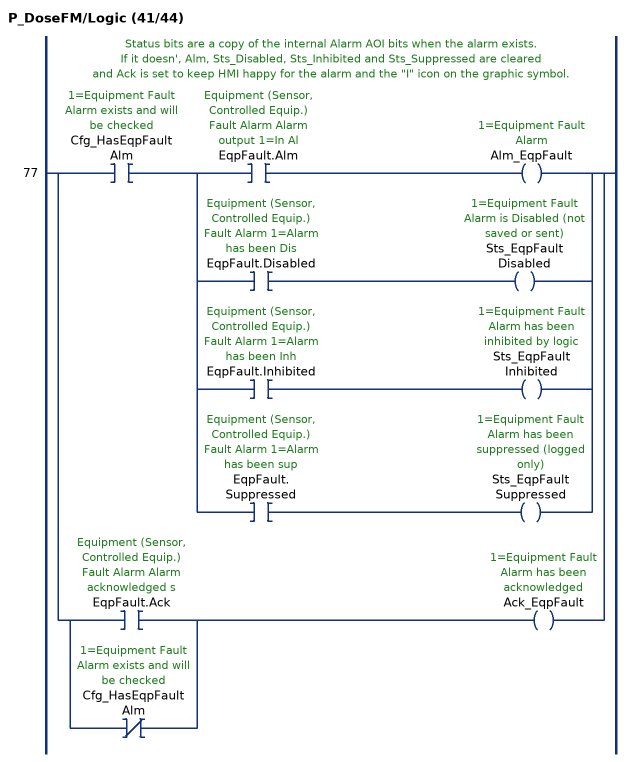
   // Status bits are a copy of the internal Alarm AOI bits when the alarm exists.
   // If it doesn', Alm, Sts_Disabled, Sts_Inhibited and Sts_Suppressed are cleared
   // and Ack is set to keep HMI happy for the alarm and the "I" icon on the graphic symbol.
   77: [XIC(Cfg_HasEqpFaultAlm) [XIC(EqpFault.Alm) OTE(Alm_EqpFault) ,XIC(EqpFault.Disabled) OTE(Sts_EqpFaultDisabled) ,XIC(EqpFault.Inhibited) OTE(Sts_EqpFaultInhibited) ,XIC(EqpFault.Suppressed) OTE(Sts_EqpFaultSuppressed) ] ,[XIC(EqpFault.Ack) ,XIO(Cfg_HasEqpFaultAlm) ] OTE(Ack_EqpFault) ];
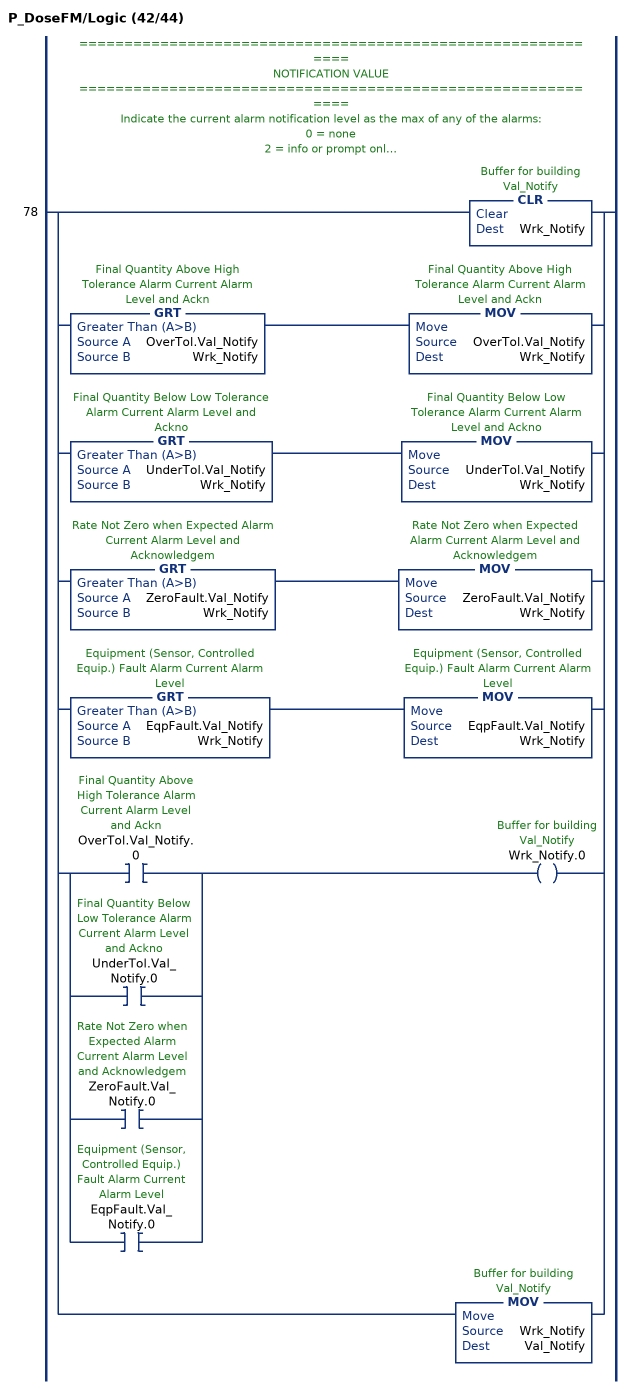
   // ============================================================
   // NOTIFICATION VALUE
   // ============================================================
   // Indicate the current alarm notification level as the max of any of the alarms:
   // 0 = none
   // 2 = info or prompt only
   // 4 = warning
   // 6 = exception (equipment impact)
   // 8 = fault (equipment failure)
   // Add one for any unsuppressed alarm that is not acknowledged (for blink).
   78: [CLR(Wrk_Notify) ,GRT(OverTol.Val_Notify,Wrk_Notify) MOV(OverTol.Val_Notify,Wrk_Notify) ,GRT(UnderTol.Val_Notify,Wrk_Notify) MOV(UnderTol.Val_Notify,Wrk_Notify) ,GRT(ZeroFault.Val_Notify,Wrk_Notify) MOV(ZeroFault.Val_Notify,Wrk_Notify) ,GRT(EqpFault.Val_Notify,Wrk_Notify) MOV(EqpFault.Val_Notify,Wrk_Notify) ,[XIC(OverTol.Val_Notify.0) ,XIC(UnderTol.Val_Notify.0) ,XIC(ZeroFault.Val_Notify.0) ,XIC(EqpFault.Val_Notify.0) ] OTE(Wrk_Notify.0) ,MOV(Wrk_Notify,Val_Notify) ];
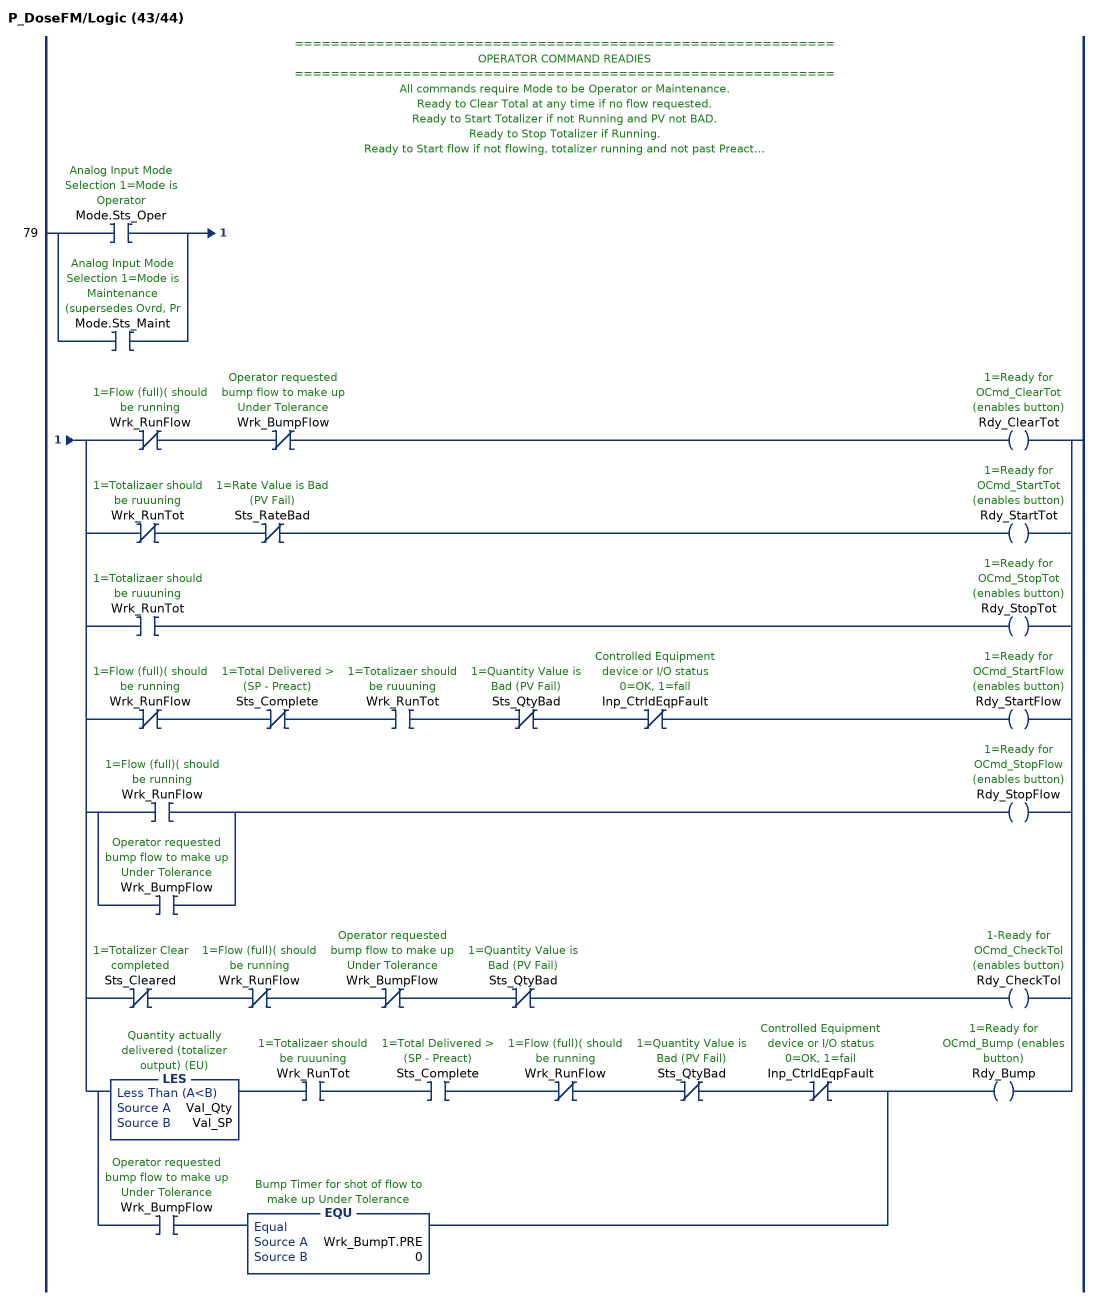
   // ============================================================
   // OPERATOR COMMAND READIES
   // ============================================================
   // All commands require Mode to be Operator or Maintenance.
   // Ready to Clear Total at any time if no flow requested.
   // Ready to Start Totalizer if not Running and PV not BAD.
   // Ready to Stop Totalizer if Running.
   // Ready to Start flow if not flowing, totalizer running and not past Preact.
   // Ready to Stop flow if flowing or in bump.
   // Ready to Check Tolerances if PV is not BAD and not flowing.
   // Ready to bump if PV not BAD, past preact but not complete, totalizer is running, and not flowing.
   // NOTE:  Keep the BUMP button active as long as a bump is in progress if
   // the Bump Time is 0 -- this keeps the button on-screen so the bump command is
   // cleared if the operator releases the button!!!
   79: [XIC(Mode.Sts_Oper) ,XIC(Mode.Sts_Maint) ][XIO(Wrk_RunFlow) XIO(Wrk_BumpFlow) OTE(Rdy_ClearTot) ,XIO(Wrk_RunTot) XIO(Sts_RateBad) OTE(Rdy_StartTot) ,XIC(Wrk_RunTot) OTE(Rdy_StopTot) ,XIO(Wrk_RunFlow) XIO(Sts_Complete) XIC(Wrk_RunTot) XIO(Sts_QtyBad) XIO(Inp_CtrldEqpFault) OTE(Rdy_StartFlow) ,[XIC(Wrk_RunFlow) ,XIC(Wrk_BumpFlow) ] OTE(Rdy_StopFlow) ,XIO(Sts_Cleared) XIO(Wrk_RunFlow) XIO(Wrk_BumpFlow) XIO(Sts_QtyBad) OTE(Rdy_CheckTol) ,[LES(Val_Qty,Val_SP) XIC(Wrk_RunTot) XIC(Sts_Complete) XIO(Wrk_RunFlow) XIO(Sts_QtyBad) XIO(Inp_CtrldEqpFault) ,XIC(Wrk_BumpFlow) EQU(Wrk_BumpT.PRE,0) ] OTE(Rdy_Bump) ];
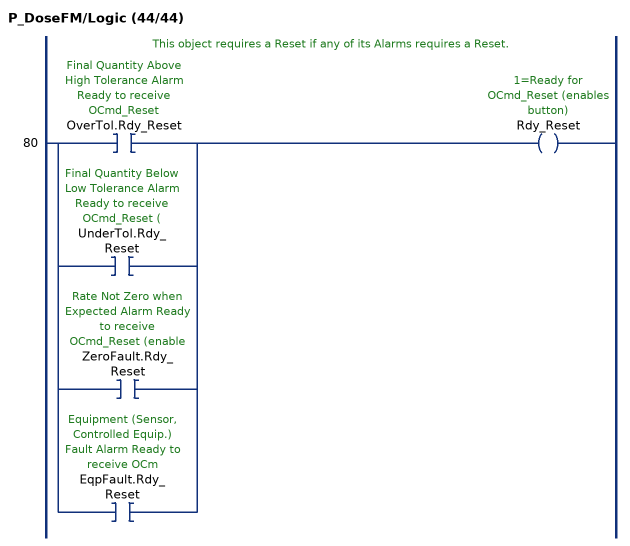
   // This object requires a Reset if any of its Alarms requires a Reset.
   80: [XIC(OverTol.Rdy_Reset) ,XIC(UnderTol.Rdy_Reset) ,XIC(ZeroFault.Rdy_Reset) ,XIC(EqpFault.Rdy_Reset) ]OTE(Rdy_Reset);
END_ROUTINE
